FUNCTION_BLOCK FB_PumpTransportTube EXTENDS FB_Operation
VAR_INPUT
END_VAR
VAR_OUTPUT
END_VAR
VAR
END_VAR

SUPER^();

END_FUNCTION_BLOCK

(* stored: Version 1.1.0.1, ProductVersion 3.1.4024.0
   POU FB_PumpTransportTube: Id {18af31ad-0ef4-4293-b083-bfbe97dbfcd2}, SpecialFunc None *)
